TYPE ST_Machine_Cfg :
	STRUCT
	END_STRUCT
END_TYPE

(* stored: Version 1.1.0.1
   DUT ST_Machine_Cfg: Id {fa4f7889-36ae-4ab3-a2fc-328e38f91015} *)
